{attribute 'GeneratedUsingTerminal: EL3403-0000-0018'}
{attribute addProperty BoxType "EL3403-0000-0018"}
{attribute addProperty Id "EtcSlaveTerminalBasePM_Inputs_Channel_1AT %I*PM_Inputs_Channel_2468BF1D19PM_Inputs_Channel_2AT %I*PM_Inputs_Channel_2468BF1D19PM_Inputs_Channel_3AT %I*PM_Inputs_Channel_2468BF1D19PM_Status_dataAT %I*PM_Status_data_0FD072A05PM_Outputs_Channel_1AT %Q*PM_Outputs_Channel_E5FBDE301PM_Outputs_Channel_2AT %Q*PM_Outputs_Channel_E5FBDE301PM_Outputs_Channel_3AT %Q*PM_Outputs_Channel_E5FBDE301WcStateAT %I*WcState_9091E0EB2InfoDataAT %I*InfoData_32EB74EA10"}
{attribute addProperty CRC "608360527"}
{attribute addProperty Size "77"}
TYPE EL3403_2442D84F EXTENDS EtcSlaveTerminalBase :
STRUCT
	{attribute addProperty Name "PM_Inputs_Channel_1"}
	PM_Inputs_Channel_1 : PM_Inputs_Channel_2468BF1D;
	{attribute addProperty Name "PM_Inputs_Channel_2"}
	PM_Inputs_Channel_2 : PM_Inputs_Channel_2468BF1D;
	{attribute addProperty Name "PM_Inputs_Channel_3"}
	PM_Inputs_Channel_3 : PM_Inputs_Channel_2468BF1D;
	{attribute addProperty Name "PM_Status_data"}
	PM_Status_data : PM_Status_data_0FD072A0;
	{attribute addProperty Name "PM_Outputs_Channel_1"}
	PM_Outputs_Channel_1 : PM_Outputs_Channel_E5FBDE30;
	{attribute addProperty Name "PM_Outputs_Channel_2"}
	PM_Outputs_Channel_2 : PM_Outputs_Channel_E5FBDE30;
	{attribute addProperty Name "PM_Outputs_Channel_3"}
	PM_Outputs_Channel_3 : PM_Outputs_Channel_E5FBDE30;
	{attribute addProperty Name "WcState"}
	WcState : WcState_9091E0EB;
	{attribute addProperty Name "InfoData"}
	InfoData : InfoData_32EB74EA;
END_STRUCT
END_TYPE

(* stored: Version 1.2.0.0, ProductVersion 3.1.4024.9
   DUT EL3403_2442D84F: Id {3e34b23a-b6db-4783-bf8a-53550aa1d7ca} *)
